// TIA Portal V19 export
TYPE "LUC_typeDiagnostics"
TITLE = LUC_typeStateModeManagerDiagnostics
// Module related diagnostic information
// stored: Access Published
   STRUCT
      interfaceManagerStatus { ExternalWritable := 'False'} : Word;   // Status of the FB InterfaceManager / Actual buffer Entry
      modeStateManagerDiagnostics { ExternalWritable := 'False'} : "LPMLV2022_typeDiagnostics";   // Diagnostics of the FB UnitModeStateManager
   END_STRUCT;
END_TYPE
